ABB RobotStudio station: Practica2Avanzada2_EstacionDePartida_1.rspag

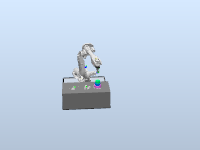
--- station ---
Station Practica2Avanzada2_EstacionDePartida_1 (saved by RobotStudio 20.4.9280.0)
Controller Sistema6
  mechanical unit ROB_1: IRB6640_180_255__04, 6 joints, base frame (0, 0, 0) mm
Layout (positions relative to the parent item):
  - Ventosa [mechanism] at (1500, 500, 1650) mm, rotated rx -180 ry 0 rz -180 deg
      TCP Ventosa at (0, 0, 200) mm
      links: PiezaVentosa
  - IRB6640_180_255__04 [mechanism, from Robots\IRB6640_180_255_G_04.rslib] at (0, 0, 0) mm; joint values [0.3218, 0.0943, 0.0791, 0, 1.3973, 0.3218] (rad or m)
  - MesaTrabajoParteIzq [part]
  - MesaTrabajoParteDer [part]
  - CI_VentosaVacuostato [smart component]
      signals: DI ActivaVentosa, DO Vacuostato
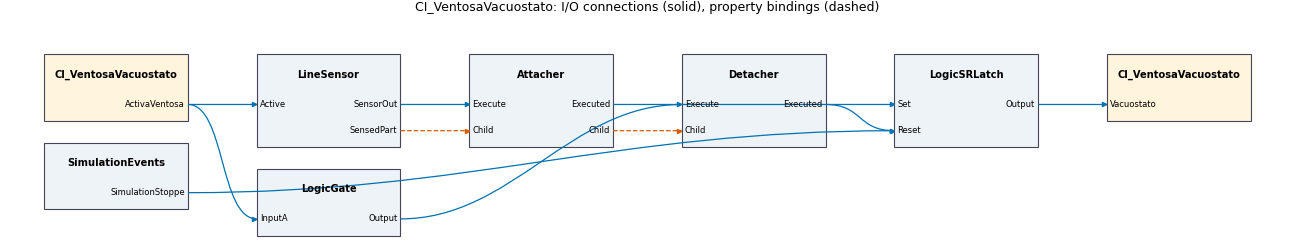
      connections:
        CI_VentosaVacuostato.ActivaVentosa -> LineSensor.Active
        LineSensor.SensorOut -> Attacher.Execute
        Attacher.Executed -> LogicSRLatch.Set
        LogicSRLatch.Output -> CI_VentosaVacuostato.Vacuostato
        Detacher.Executed -> LogicSRLatch.Reset
        SimulationEvents.SimulationStopped -> LogicSRLatch.Reset
        CI_VentosaVacuostato.ActivaVentosa -> LogicGate.InputA
        LogicGate.Output -> Detacher.Execute
        LineSensor.SensedPart => Attacher.Child
        Attacher.Child => Detacher.Child
    - LineSensor [smart component, from Components\LineSensor.rslib] at (1500, 500, 1450) mm, rotated rx -180 ry 0 rz -180 deg
        properties: Start=[0 0 -0.002]; End=[0 0 0.02]; Radius=0.002; SensedPart=(none); SensedPoint=[0 0 0]
      - _sensorPart_ [part]
    - SimulationEvents [smart component, from Components\SimulationEvents.rslib]
    - LogicSRLatch [smart component, from Components\LogicSRLatch.rslib]
    - Attacher [smart component, from Components\Attacher.rslib]
        properties: Parent=Ventosa; Flange=0; Child=(none); Mount=false; Offset=[0 0 0]; Orientation=[0 0 0]
    - Detacher [smart component, from Components\Detacher.rslib]
        properties: Child=(none); KeepPosition=true
    - LogicGate [smart component, from Components\LogicGate.rslib]
        properties: Operator=NOT; Delay=0.1
  - BaseOrigen [part]
  - BaseDestino [part]
  - BaseInterm [part]
  - Pieza_1 [part]
  - Pieza_2 [part]
  - Pieza_3 [part]
Attachment: LineSensor is attached to Ventosa / PiezaVentosa
Attachment: Ventosa is attached to IRB6640_180_255__04 / Link6
Station logic (signal -> signal, property => property):
  CI_VentosaVacuostato.Vacuostato -> Sistema6.ED_PiezaCogida
  Sistema6.SD_ActivaVentosa -> CI_VentosaVacuostato.ActivaVentosa

--- Backups/Sistema6/RAPID/TASK1/PROGMOD/CalibData.mod ---
MODULE CalibData
	PERS tooldata Ventosa:=[TRUE,[[0,0,200],[1,0,0,0]],[1,[0,0,125],[1,0,0,0],0.002,0.002,0.0013]];
ENDMODULE

--- Backups/Sistema6/RAPID/TASK1/PROGMOD/Module1.mod ---
MODULE Module1
	CONST robtarget pReposo:=[[1808.910161514,0,1855],[0.5,0,0.866025404,0],[0,0,0,0],[9E+09,9E+09,9E+09,9E+09,9E+09,9E+09]];
	CONST robtarget pBaseTorre1:=[[1500,500,750],[0,0,1,0],[0,0,0,0],[9E+09,9E+09,9E+09,9E+09,9E+09,9E+09]];
    CONST robtarget pBaseTorre2:=[[1500,-500,750],[0,0,1,0],[0,0,0,0],[9E+09,9E+09,9E+09,9E+09,9E+09,9E+09]];
    CONST robtarget pBaseDestino:=[[1500,-500,750],[0,0,1,0],[0,0,0,0],[9E+09,9E+09,9E+09,9E+09,9E+09,9E+09]];
    CONST robtarget pBaseInterm:=[[1500,0,750],[0,0,1,0],[0,0,0,0],[9E+09,9E+09,9E+09,9E+09,9E+09,9E+09]];
    CONST robtarget pBaseOrigen:=[[1500,500,750],[0,0,1,0],[0,0,0,0],[9E+09,9E+09,9E+09,9E+09,9E+09,9E+09]];

    CONST num altura := 100;
    CONST num nPiezasTotales := 3;
    VAR num alturaOrigen := nPiezasTotales * altura;
    VAR num alturaDestino := altura;
    VAR num alturaInter := altura;


    PROC main()
        VAR robtarget pOrig;
        pOrig := Offs (pBaseOrigen, 0, 0, (nPiezasTotales * altura) + altura);
        TorresHanoi nPiezasTotales, pOrig, pBaseDestino, pBaseInterm, altura;
    ENDPROC

    PROC TorresHanoi (num nPiezas, robtarget pOrig, robtarget pDest, robtarget pInt, num altoPieza)

        VAR robtarget pAproxOrigen;
        VAR robtarget pAproxDestino;
        VAR robtarget pAproxInter;
        VAR robtarget pAux1;
        VAR robtarget pAux2;

        !Definimos los puntos de aproximación
        pAproxOrigen := Offs (pOrig, 0, 0, altura * nPiezasTotales + altura);
        pAproxDestino := Offs (pDest, 0, 0, altura * nPiezasTotales + altura);
        pAproxInter := Offs (pInt, 0, 0, altura * nPiezasTotales + altura);

        IF nPiezas = 1 THEN

            !Movemos la pieza del origen al destino
            MoveL pAproxOrigen, v2000, fine,Ventosa\WObj:=wobj0;
            MoveLDO pOrig, v2000, fine,Ventosa\WObj:=wobj0, SD_ActivaVentosa, 1;
            WaitDI ED_PiezaCogida, 1;

            MoveL pAproxDestino, v2000, fine,Ventosa\WObj:=wobj0;
            MoveLDO pDest, v2000, fine,Ventosa\WObj:=wobj0, SD_ActivaVentosa, 0;
            WaitDI ED_PiezaCogida, 0;

        ELSE

            !Hacemos Hanoi(n-1, origen, destino, auxiliar)
            pOrig := Offs (pOrig, 0, 0, -altura);
            pDest := Offs (pDest, 0, 0, altura * nPiezas);
            pInt := Offs (pInt, 0, 0, 0);
            TorresHanoi nPiezas - 1, pOrig, pInt, pDest, altoPieza;

            !Movemos la pieza del origen al destino
            pOrig := Offs (pOrig, 0, 0, altura * nPiezas);
            pDest := Offs (pDest, 0, 0, -altura);
            pInt := Offs (pInt, 0, 0, 0);
            MoveL pAproxOrigen, v2000, fine,Ventosa\WObj:=wobj0;
            MoveLDO pOrig, v2000, fine,Ventosa\WObj:=wobj0, SD_ActivaVentosa, 1;
            WaitDI ED_PiezaCogida, 1;

            MoveL pAproxDestino, v2000, fine,Ventosa\WObj:=wobj0;
            MoveLDO pDest, v2000, fine,Ventosa\WObj:=wobj0, SD_ActivaVentosa, 0;
            WaitDI ED_PiezaCogida, 0;


            !Hacemos Hanoi(n-1, auxiliar, origen, destino)
            TorresHanoi nPiezas - 1, pInt, pDest, pOrig, altoPieza;

        ENDIF

    ENDPROC

ENDMODULE

--- Backups/Sistema6/RAPID/TASK1/SYSMOD/LINKEDM.sys ---
%%%
  VERSION:1
  LANGUAGE:ENGLISH
%%%

MODULE LINKEDM (SYSMODULE)

! FOLLOWER
!     Name of electronically linked follower axis used by operator at teach pendent.
      PERS string l_f_axis_name{5}       :=  ["",  "", "", "", ""];

!     Name of the mechanical unit for follower axis.
      PERS string l_f_mecunt_n{5}  :=  ["", "", "", "", ""];

!     Linked follower axis number in the mechanical unit (first axis in mech. unit is number 1).
      PERS num l_f_axis_no{5}      :=  [0,          0,   0,  0,  0];

! MASTER
!     Name of the mechanical unit for linked master axis.
      PERS string l_m_mecunt_n{5} :=  ["", "", "", "", ""];

!     Linked master axis number in the mechanical unit (first axis in mech. unit is number 1).
!     See axis number table in documentation for different master mechanical units.
      PERS num l_m_axis_no{5}     :=  [0,  0,  0,  0,  0];

! POSITION OFFSET
!     The increase of the allowed offset position between the master and follower
!     positions, used when starting AUTO mode. As soon as the offset is decreased
!     the old configurated parameter is used.
!     Example: 3 => the configurated value of allowed offset is increased 3 times.
      PERS num offset_ratio{5}       :=  [10,  10,   10,  10,  10];

! SPEED RATIO
!     Speed_ratio used in AUTO and JOG modes [ very_slow   slow    normal    fast]
!     Value 1 = max allowed manual speed.
      CONST num speed_ratio {20}      := [0.01, 0.01, 0.01, 0.01, 0.01,
                                          0.05, 0.05, 0.05, 0.05, 0.05,
                                          0.20, 0.20, 0.20, 0.20, 0.20,
                                          1.00, 1.00, 1.00, 1.00, 1.00];

! STEP SIZE
!     Displacement position used in JOG mode for each activation of positive or
!     negative movement.                  [very_short    short   normal   long]
!     Unit degees or meter.
      CONST num displacement {20}     := [0.001, 0.001, 0.001, 0.001, 0.001,
                                          0.005, 0.005, 0.005, 0.005, 0.005,
                                          0.020, 0.020, 0.020, 0.020, 0.020,
                                          0.100, 0.100, 0.100, 0.100, 0.100];


!-------------------------------------------------------------
 PROC Linked_m ()
      Linked_m_exe ;
 ENDPROC
ENDMODULE

--- Backups/Sistema6/SYSPAR/EIO.cfg ---
EIO:CFG_1.0:6:1::
#
INDUSTRIAL_NETWORK:

      -Name "DeviceNet" -Label "DeviceNet Master/Slave Network" -Address "2"
#
DEVICENET_DEVICE:

      -Name "MiDeviceNet" -Label "MiDeviceNet"
#
DEVICENET_INTERNAL_DEVICE:

      -Name "DN_Internal_Device" -VendorName "ABB Robotics"\
      -ProductName "DeviceNet Internal Slave Device"
#
EIO_SIGNAL:

      -Name "ED_PiezaCogida" -SignalType "DI" -Device "MiDeviceNet"\
      -Label "ED_PiezaCogida" -DeviceMap "0" -Access "All"

      -Name "SD_ActivaVentosa" -SignalType "DO" -Device "MiDeviceNet"\
      -Label "SD_ActivaVentosa" -DeviceMap "0" -Access "All"
